{attribute 'qualified_only'}
{attribute 'strict'}
{attribute 'to_string'}
TYPE ObjectState :
(
	AUS 			:= 0,				// Das Objekt ist ausgeschalten
	BEREIT 			:= 1,				// Das Objekt ist eingeschalten und bereit
	LAUFEND 		:= 2,				// Das Objekt ist aktiv
	ABGESCHLOSSEN 	:= 3,				// Das Objekt hat den Prozess durchgeführt und hat selbständig gestoppt
	GESTOPPT 		:= 4,				// Das Objekt wurde gestoppt durch externe Einwirkung gestoppt
	FEHLER			:= 5				// Es gibt einen Fehler bezüglich des Objektes
);
END_TYPE

(* stored: Version 1.1.0.1
   DUT ObjectState: Id {706355d0-793c-4252-b246-a24d3f27e796} *)
